TYPE "InfeedAlr"
VERSION : 0.1
// Block: InfeedAlr
   STRUCT
      InfeedFault : Bool;
      ComunicationFault : Bool;
      TimeoutActivation : Bool;
      GeneralError : Bool;
   END_STRUCT;

END_TYPE
